// TwinCAT 3 PLC project
// project tree:
//   POUs/ MAIN.TcPOU
//   DUTs/ timer_location.TcDUT, sup_location.TcDUT, hw_button_location.TcDUT, hw_lamp_location.TcDUT
//   GVLs/ INPUTS.TcGVL, OUTPUTS.TcGVL, TIMERS.TcGVL

// ---- DUTs/timer_location.TcDUT
TYPE timer_location:
    (timer_Idle, timer_Running);
END_TYPE

// ---- DUTs/sup_location.TcDUT
TYPE sup_location:
    (s1_sup_location, s2_sup_location, s3_sup_location, s4_sup_location, s5_sup_location, s6_sup_location, s7_sup_location, s8_sup_location, s9_sup_location, s10_sup_location);
END_TYPE

// ---- DUTs/hw_button_location.TcDUT
TYPE hw_button_location:
    (Released_hw_button_location, Pushed_hw_button_location);
END_TYPE

// ---- DUTs/hw_lamp_location.TcDUT
TYPE hw_lamp_location:
    (hw_lamp_Off, hw_lamp_On);
END_TYPE

// ---- GVLs/INPUTS.TcGVL
VAR_GLOBAL // INPUTS
    in_hw_button_bit AT %I15.5: BOOL;
    in_hw_button_bot AT %I18: DINT;
    in_hw_button_bat AT %I19: REAL;
END_VAR

// ---- GVLs/OUTPUTS.TcGVL
VAR_GLOBAL // OUTPUTS
    out_hw_lamp_bit AT %Q16.6: BOOL;
END_VAR

// ---- GVLs/TIMERS.TcGVL
VAR_GLOBAL // TIMERS
    ton_timer_t: TON;
END_VAR

// ---- POUs/MAIN.TcPOU
PROGRAM MAIN
VAR
    timer_t: LREAL;
    preset_timer_t: TIME;
    timer: timer_location;
    sup: sup_location;
    hw_button_bit: BOOL;
    hw_button: hw_button_location;
    hw_lamp_bit: BOOL;
    hw_lamp: hw_lamp_location;
    firstRun: BOOL := TRUE;
END_VAR
VAR_TEMP
    curValue: LREAL;
    current_hw_button: hw_button_location;
    current_hw_button__1: hw_button_location;
    current_hw_lamp: hw_lamp_location;
    current_hw_lamp__1: hw_lamp_location;
    current_hw_lamp_bit: BOOL;
    current_hw_lamp_bit__1: BOOL;
    current_sup: sup_location;
    current_sup__1: sup_location;
    current_sup__2: sup_location;
    current_sup__3: sup_location;
    current_sup__4: sup_location;
    current_sup__5: sup_location;
    current_timer: timer_location;
    current_timer__1: timer_location;
    current_timer_t: LREAL;
    eventEnabled: BOOL;
    isProgress: BOOL;
    syncAutEdge: DINT;
    syncAutEdge__1: DINT;
    syncAutEdge__10: DINT;
    syncAutEdge__11: DINT;
    syncAutEdge__2: DINT;
    syncAutEdge__3: DINT;
    syncAutEdge__4: DINT;
    syncAutEdge__5: DINT;
    syncAutEdge__6: DINT;
    syncAutEdge__7: DINT;
    syncAutEdge__8: DINT;
    syncAutEdge__9: DINT;
    timeOut: BOOL;
END_VAR

(* --- Read input from sensors. -------------------------------------------- *)
hw_button_bit := in_hw_button_bit;

(* --- Initialize state or update continuous variables. -------------------- *)
IF firstRun THEN
    firstRun := FALSE;

    (* Initialize the state variables. *)
    timer_t := 0.0;
    (* Reset timer of "timer_t". *)
    preset_timer_t := timer_t;
    ton_timer_t(IN := FALSE, PT := preset_timer_t);
    ton_timer_t(IN := TRUE, PT := preset_timer_t);
    timer := timer_Idle;
    sup := sup_s1;
    hw_button := hw_button_Released;
    hw_lamp_bit := FALSE;
    hw_lamp := hw_lamp_Off;
ELSE
    (* Update remaining time of "timer_t". *)
    ton_timer_t(IN := TRUE, PT := preset_timer_t, Q => timeOut, ET => curValue);
    timer_t := SEL(timeOut, preset_timer_t - curValue, 0.0);
END_IF;

(* --- Process all events. ------------------------------------------------- *)
isProgress := TRUE;
(* Perform events until none can be done anymore. *)
WHILE isProgress DO
    isProgress := FALSE;

    (* Try to perform event "timer.start". *)
    eventEnabled := TRUE;
    IF timer = timer_Idle THEN
        syncAutEdge := 1;
    ELSE
        eventEnabled := FALSE;
    END_IF;
    IF eventEnabled THEN
        IF sup = sup_s3 THEN
            syncAutEdge__1 := 1;
        ELSIF sup = sup_s5 THEN
            syncAutEdge__1 := 2;
        ELSE
            eventEnabled := FALSE;
        END_IF;
    END_IF;
    IF eventEnabled THEN
        isProgress := TRUE;
        current_sup := sup;
        current_timer := timer;
        current_timer_t := timer_t;
        IF syncAutEdge = 1 THEN
            timer_t := 3.0;
            (* Reset timer of "timer_t". *)
            preset_timer_t := timer_t;
            ton_timer_t(IN := FALSE, PT := preset_timer_t);
            ton_timer_t(IN := TRUE, PT := preset_timer_t);
            timer := timer_Running;
        END_IF;
        IF syncAutEdge__1 = 1 THEN
            sup := sup_s6;
        ELSIF syncAutEdge__1 = 2 THEN
            sup := sup_s7;
        END_IF;
    END_IF;

    (* Try to perform event "timer.timeout". *)
    eventEnabled := TRUE;
    IF timer = timer_Running AND timer_t <= 0.0 THEN
        syncAutEdge__2 := 1;
    ELSE
        eventEnabled := FALSE;
    END_IF;
    IF eventEnabled THEN
        IF sup = sup_s6 THEN
            syncAutEdge__3 := 1;
        ELSIF sup = sup_s7 THEN
            syncAutEdge__3 := 2;
        ELSE
            eventEnabled := FALSE;
        END_IF;
    END_IF;
    IF eventEnabled THEN
        isProgress := TRUE;
        current_sup__1 := sup;
        current_timer__1 := timer;
        IF syncAutEdge__2 = 1 THEN
            timer := timer_Idle;
        END_IF;
        IF syncAutEdge__3 = 1 THEN
            sup := sup_s8;
        ELSIF syncAutEdge__3 = 2 THEN
            sup := sup_s9;
        END_IF;
    END_IF;

    (* Try to perform event "button.push". *)
    eventEnabled := TRUE;
    IF sup = sup_s1 THEN
        syncAutEdge__4 := 1;
    ELSIF sup = sup_s4 THEN
        syncAutEdge__4 := 2;
    ELSIF sup = sup_s5 THEN
        syncAutEdge__4 := 3;
    ELSIF sup = sup_s7 THEN
        syncAutEdge__4 := 4;
    ELSIF sup = sup_s9 THEN
        syncAutEdge__4 := 5;
    ELSE
        eventEnabled := FALSE;
    END_IF;
    IF eventEnabled THEN
        IF hw_button = hw_button_Released AND hw_button_bit THEN
            syncAutEdge__5 := 1;
        ELSE
            eventEnabled := FALSE;
        END_IF;
    END_IF;
    IF eventEnabled THEN
        isProgress := TRUE;
        current_hw_button := hw_button;
        current_sup__2 := sup;
        IF syncAutEdge__4 = 1 THEN
            sup := sup_s2;
        ELSIF syncAutEdge__4 = 2 THEN
            sup := sup_s2;
        ELSIF syncAutEdge__4 = 3 THEN
            sup := sup_s3;
        ELSIF syncAutEdge__4 = 4 THEN
            sup := sup_s6;
        ELSIF syncAutEdge__4 = 5 THEN
            sup := sup_s8;
        END_IF;
        IF syncAutEdge__5 = 1 THEN
            hw_button := hw_button_Pushed;
        END_IF;
    END_IF;

    (* Try to perform event "button.release". *)
    eventEnabled := TRUE;
    IF sup = sup_s2 THEN
        syncAutEdge__6 := 1;
    ELSIF sup = sup_s3 THEN
        syncAutEdge__6 := 2;
    ELSIF sup = sup_s6 THEN
        syncAutEdge__6 := 3;
    ELSIF sup = sup_s8 THEN
        syncAutEdge__6 := 4;
    ELSIF sup = sup_s10 THEN
        syncAutEdge__6 := 5;
    ELSE
        eventEnabled := FALSE;
    END_IF;
    IF eventEnabled THEN
        IF hw_button = hw_button_Pushed AND NOT hw_button_bit THEN
            syncAutEdge__7 := 1;
        ELSE
            eventEnabled := FALSE;
        END_IF;
    END_IF;
    IF eventEnabled THEN
        isProgress := TRUE;
        current_hw_button__1 := hw_button;
        current_sup__3 := sup;
        IF syncAutEdge__6 = 1 THEN
            sup := sup_s4;
        ELSIF syncAutEdge__6 = 2 THEN
            sup := sup_s5;
        ELSIF syncAutEdge__6 = 3 THEN
            sup := sup_s7;
        ELSIF syncAutEdge__6 = 4 THEN
            sup := sup_s9;
        ELSIF syncAutEdge__6 = 5 THEN
            sup := sup_s1;
        END_IF;
        IF syncAutEdge__7 = 1 THEN
            hw_button := hw_button_Released;
        END_IF;
    END_IF;

    (* Try to perform event "lamp.on". *)
    eventEnabled := TRUE;
    IF sup = sup_s2 THEN
        syncAutEdge__8 := 1;
    ELSIF sup = sup_s4 THEN
        syncAutEdge__8 := 2;
    ELSE
        eventEnabled := FALSE;
    END_IF;
    IF eventEnabled THEN
        IF hw_lamp = hw_lamp_Off THEN
            syncAutEdge__9 := 1;
        ELSE
            eventEnabled := FALSE;
        END_IF;
    END_IF;
    IF eventEnabled THEN
        isProgress := TRUE;
        current_hw_lamp := hw_lamp;
        current_hw_lamp_bit := hw_lamp_bit;
        current_sup__4 := sup;
        IF syncAutEdge__8 = 1 THEN
            sup := sup_s3;
        ELSIF syncAutEdge__8 = 2 THEN
            sup := sup_s5;
        END_IF;
        IF syncAutEdge__9 = 1 THEN
            hw_lamp_bit := TRUE;
            hw_lamp := hw_lamp_On;
        END_IF;
    END_IF;

    (* Try to perform event "lamp.off". *)
    eventEnabled := TRUE;
    IF sup = sup_s8 THEN
        syncAutEdge__10 := 1;
    ELSIF sup = sup_s9 THEN
        syncAutEdge__10 := 2;
    ELSE
        eventEnabled := FALSE;
    END_IF;
    IF eventEnabled THEN
        IF hw_lamp = hw_lamp_On THEN
            syncAutEdge__11 := 1;
        ELSE
            eventEnabled := FALSE;
        END_IF;
    END_IF;
    IF eventEnabled THEN
        isProgress := TRUE;
        current_hw_lamp__1 := hw_lamp;
        current_hw_lamp_bit__1 := hw_lamp_bit;
        current_sup__5 := sup;
        IF syncAutEdge__10 = 1 THEN
            sup := sup_s10;
        ELSIF syncAutEdge__10 = 2 THEN
            sup := sup_s1;
        END_IF;
        IF syncAutEdge__11 = 1 THEN
            hw_lamp_bit := FALSE;
            hw_lamp := hw_lamp_Off;
        END_IF;
    END_IF;
END_WHILE;

(* --- Write output to actuators. ------------------------------------------ *)
out_hw_lamp_bit := hw_lamp_bit;

END_PROGRAM
